FUNCTION_BLOCK FB_HMI_METIS_CTRL_TEMPERATURE EXTENDS FB_HMI_COMPONENT
VAR_INPUT
END_VAR
VAR_OUTPUT
END_VAR
VAR_IN_OUT
    fbInstance : FB_METIS_CTRL_TEMPERATURE;
END_VAR
VAR
END_VAR

fbHealthStatus(
    bIsEnabled := fbInstance.cfg.bEnabled,
    bIsGood := fbInstance.stat.bValid);
                     
fbBusyStatus(
    bIsEnabled := FALSE,
    bIsBusy := FALSE);

M_UpdateStatusColor();

END_FUNCTION_BLOCK

(* stored: Version 1.1.0.1, ProductVersion 3.1.4024.14
   POU FB_HMI_METIS_CTRL_TEMPERATURE: Id {4854d037-6920-4e91-a716-a489f8ae3eaa}, SpecialFunc None *)
